///automatically generated by the FlatBuffers compiler, do not modify
///comm\datalayer
{attribute 'conditionalshow' := ''}
METHOD verifyProgressData : BOOL
VAR_INPUT
	data: POINTER TO BYTE;
	size: __UXINT;
	pointer_: UDINT;
END_VAR
VAR
	_bb: ByteBuffer;
	verifier: flatbuffers.Verifier;
	vt_start: UDINT;
	vt_size: UDINT;
END_VAR
_bb(data:=data, _capacity:=TO_UDINT(size));
IF pointer_ = 0 THEN
    verifyProgressData := TRUE;
    RETURN;
END_IF

if pointer_ > (size - SIZEOF(UDINT)) then
    verifyProgressData := FALSE;
    return;
END_IF

vt_start := _bb.getUDINT(pointer_);
if (pointer_ - vt_start) > (size - SIZEOF(UDINT)) then
    verifyProgressData := FALSE;
    return;
END_IF

vt_size := _bb.getUINT(pointer_ - vt_start);
verifier(data:=data, size:=size, pointer_:=pointer_, v_size:=vt_size);

IF verifier.verifyTable() AND verifier.verifyString(4) AND verifier.verifyString(6) THEN
    verifyProgressData := TRUE;
ELSE
    verifyProgressData := FALSE;
END_IF
END_METHOD

END_FUNCTION_BLOCK

// InternHelpers/DCBrowseForFile
{attribute 'hide'}
FUNCTION_BLOCK DCBrowseForFile
VAR_INPUT
	bExecute: BOOL;
	sFileName: STRING;
END_VAR
VAR_OUTPUT
	bDone: BOOL;
	bActive: BOOL;
	bError: BOOL;
	bFound: BOOL;
	ErrorID: CXA_Datalayer.ERROR_CODE;
	ErrorIdent: CXA_Datalayer.ERROR_STRUCT;
END_VAR
VAR
	_dlBrowse: CXA_DATALAYER.DL_BrowseNode;
	_sPath: STRING := S_PARAM_PATH;
	_uiState: UINT;
	_uiNextState: UINT;
	_i: UDINT;
END_VAR
VAR CONSTANT
	S_PARAM_PATH: STRING := 'driveconnect/filesystem/parameterfiles';
	STATE_IDLE: UINT := 0;
	STATE_BROWSE: UINT := 1;
	STATE_CHECK: UINT := 2;
	STATE_DONE: UINT := 3;
	STATE_ERROR: UINT := 4;
END_VAR

CASE _uiState OF 
	STATE_IDLE: 
		IF bExecute THEN 
			_uiNextState := STATE_BROWSE; 
		END_IF
	STATE_BROWSE: 
		IF _dlBrowse.Error THEN 
			ErrorID := _dlBrowse.ErrorID; 
			ErrorIdent := _dlBrowse.ErrorIdent; 
			_uiNextState := STATE_ERROR; 
		ELSIF _dlBrowse.Done THEN 
			_uiNextState := STATE_CHECK; 
		END_IF
	STATE_CHECK: 
		_uiNextState := STATE_DONE; 
	STATE_DONE, STATE_ERROR: 
		IF NOT bExecute THEN 
			_uiNextState := STATE_IDLE; 
		END_IF
END_CASE
_uiState := _uiNextState; 
CASE _uiState OF 
	STATE_IDLE: 
		_dlBrowse.Execute := FALSE; 
		bFound := FALSE; 
	STATE_BROWSE: 
		_dlBrowse.Execute := TRUE;  
	STATE_CHECK:
		_i := 0;
		WHILE _i < _dlBrowse.ChildNum DO 
			IF sFileName = _dlBrowse.GetChildName(_i) THEN 
				bFound := TRUE; 
				EXIT; 
			END_IF
			_i := _i+1; 
		END_WHILE
END_CASE
bDone := _uiState = STATE_DONE; 
bActive := _uiState = STATE_BROWSE OR _uiState = STATE_CHECK; 
bError :=  _uiState = STATE_ERROR; 
_dlBrowse(NodeName := _sPath);

END_FUNCTION_BLOCK

// DriveParamRestore
FUNCTION_BLOCK DriveParamRestore
VAR_INPUT
	bExecute: BOOL;
	sDriveConnectName: STRING;
	iSubDevice: UINT;
	sFileName: STRING;
	iSetIndex: INT;
END_VAR
VAR_OUTPUT
	bDone: BOOL;
	bActive: BOOL;
	bError: BOOL;
	uiProgress: UDINT;
	enTaskState: comm_datalayer_ProgramTaskState;
	ErrorCause: EN_DRIVE_BACKUP_RESTORE_ERROR;
	ErrorID: CXA_Datalayer.ERROR_CODE;
	ErrorIdent: CXA_Datalayer.ERROR_STRUCT;
	sFailureInfo: STRING;
END_VAR
VAR
	_builder: Flatbuffers.FlatBufferBuilder;
	_retoreReq: comm_drive_importParameter_ImportParameter;
	_taskStatus: comm_Datalayer_ProgramTask;
	_pRespString: POINTER TO STRING(255);
	_sRespString: STRING(255);
	_dlCreateNode: CXA_DataLayer.DL_CreateNodeValue;
	_dlReadNode: CXA_DataLayer.DL_ReadNodeValue;
	_dlRestoreReq: CXA_DataLayer.DL_NodeValue;
	_dlTaskPath: CXA_DataLayer.DL_NodeValue;
	_dlTaskResp: CXA_Datalayer.DL_NodeValue;
	_uiState: UINT;
	_uiNextState: UINT;
	_enTaskState: comm_datalayer_ProgramTaskState;
	_sReqString: STRING(255);
	_sBackupFile: STRING(255);
	_uiOffset: UDINT;
	_browseForFile: DCBrowseForFile;
END_VAR
VAR CONSTANT
	STATE_IDLE: UINT := 0;
	STATE_FIND_FILE: UINT := 1;
	STATE_REQ: UINT := 2;
	STATE_RESTORING: UINT := 3;
	STATE_DONE: UINT := 4;
	STATE_ERROR: UINT := 5;
	S_PATH_DEVICES: STRING := 'devices/drives/';
	S_PATH_BACKUPS: STRING := 'filesystem/parameterfiles/';
END_VAR

CASE _uiState OF 
	STATE_IDLE: 
		IF bExecute THEN 
			_uiNextState := STATE_FIND_FILE; 
		END_IF
	STATE_FIND_FILE: 
		IF _browseForFile.bError THEN 
			ErrorID := _browseForFile.ErrorID; 
			ErrorIdent := _browseForFile.ErrorIdent; 
			ErrorCause :=EN_DRIVE_BACKUP_RESTORE_ERROR.FileBrowseFailed; 
			_uiNextState := STATE_ERROR; 
		ELSIF _browseForFile.bDone THEN 
			IF NOT _browseForFile.bFound THEN 
				ErrorCause := EN_DRIVE_BACKUP_RESTORE_ERROR.FileNotFound; 
				_uiNextState := STATE_ERROR; 
			ELSE 
				_uiNextState := STATE_REQ; 
			END_IF;  
		END_IF
	STATE_REQ: 
		IF _dlCreateNode.Error THEN 
			_uiNExtState := STATE_ERROR; 
			ErrorID := _dlCreateNode.ErrorID;
			ErrorIDent := _dlCreateNode.ErrorIdent; 
			ErrorCause := EN_DRIVE_BACKUP_RESTORE_ERROR.RequestFailed;  
		ELSIF _dlCreateNode.Done THEN 
			_uiNextState := STATE_RESTORING; 
		END_IF
	STATE_RESTORING: 
		IF _dlReadNode.Error THEN 
			_uiNextState := STATE_ERROR; 
			ErrorID := _dlReadNode.ErrorID;
			ErrorIDent := _dlReadNode.ErrorIdent; 
			ErrorCause := EN_DRIVE_BACKUP_RESTORE_ERROR.ProgressReadFailed;  
		ELSIF _dlReadNode.Done THEN 
			IF _enTaskState = comm_datalayer_ProgramTaskState.failed THEN 
				_uiNextState := STATE_ERROR; 
				ErrorID := _dlReadNode.ErrorID;
				ErrorIdent := _dlReadNode.ErrorIdent; 
				ErrorCause := EN_DRIVE_BACKUP_RESTORE_ERROR.RestoreFailed;  
				sFailureInfo := _taskStatus.getProgressInfo(); 
			ELSIF _enTaskState = comm_datalayer_ProgramTaskState.done THEN 
				_uiNextState := STATE_DONE; 
			ELSE
				_dlReadNode(Execute := FALSE); 
			END_IF
		END_IF
	STATE_DONE, STATE_ERROR: 
		IF NOT bExecute THEN 
			_uiNextState := STATE_IDLE; 
		END_IF
END_CASE
_uiState := _uiNextState; 
CASE _uiState OF 
	STATE_IDLE: 
		_dlReadNode.Execute := FALSE; 
		_dlCreateNode.Execute := FALSE; 
		_browseForFile.bExecute := FALSE; 
		sFailureInfo := 'OK'; 
		enTaskState := comm_datalayer_ProgramTaskState.done; 
		ErrorCause := EN_DRIVE_BACKUP_RESTORE_ERROR.OK; 
		uiProgress := 0; 
		
	STATE_FIND_FILE: 
		_browseForFile.sFileName := sFileName; 
		_browseForFile.bExecute := TRUE; 
				
	STATE_REQ: 
		_dlCreateNode.Execute := TRUE; 
		_builder(forceDefaults := TRUE); 
		_sBackupFile := CONCAT(S_PATH_BACKUPS,sFileName); 
		_sReqString := CONCAT(S_PATH_DEVICES,sDriveConnectName); 
		_sReqString := CONCAT(_sReqString,'/subdevices/subdevice-'); 
		_sReqString := CONCAT(_sReqString,INT_TO_STRING(iSubDevice)); 
		_sReqString := CONCAT(_sReqString,'/import-parameter'); 
		_uiOffset := _retoreReq.createImportParameter(builder := _builder,fileName := _sBackupFile, setIndex :=iSetIndex);
 		_builder.finish(_uiOffset); 
		_dlRestoreReq.SetFlatbuffer(_builder); 
	STATE_RESTORING: 
		_pRespString := _dlTaskPath.GetData(); 
		_sRespString := _pRespString^; 
		_dlReadNode.Execute := TRUE; 
END_CASE

_dlCreateNode(NodeName := _sReqString,
			  NodeValueIn := _dlRestoreReq, 
			  NodeValueOut := _dlTaskPath); 
			  
_dlReadNode(NodeName := _sRespString,
			NodeValue := _dlTaskResp); 
			
_browseForFile(); 


IF _dlReadNode.Done THEN 
	_taskStatus.getRootAsProgramTask(_dlTaskResp.GetData(),_dlTaskResp.GetSize()); 
	_enTaskState := _taskStatus.getState(); 
	uiProgress := _taskStatus.getProgress(); 
	enTaskState := _enTaskState; 
END_IF

bActive := _uiState <> STATE_IDLE AND _uiState <> STATE_DONE AND _uiState <> STATE_ERROR; 
bDone := _uiState = STATE_DONE; 
bError := _uiState = STATE_ERROR;

END_FUNCTION_BLOCK

// InternHelpers/comm_drive_importParameter_ImportParameter
///automatically generated by the FlatBuffers compiler, do not modify
///comm\drive\importParameter
///Import FlatBuffers Library
FUNCTION_BLOCK comm_drive_importParameter_ImportParameter EXTENDS flatbuffers.Table
VAR
	_builder: REFERENCE TO flatbuffers.FlatBufferBuilder;
	_bb: flatbuffers.ByteBuffer;
END_VAR

///automatically generated by the FlatBuffers compiler, do not modify
///comm\drive\importParameter
///
///Set the values of a ImportParameter and return it.
{attribute 'conditionalshow' := ''}
METHOD _assign : comm_drive_importParameter_ImportParameter
VAR_INPUT
	i: UDINT;
	_bb: REFERENCE TO flatbuffers.ByteBuffer;
END_VAR
_init(i:=i, _bb:=_bb);
_assign:=this^;
END_METHOD

///automatically generated by the FlatBuffers compiler, do not modify
///comm\drive\importParameter
///
///Set the values of a table.
{attribute 'conditionalshow' := ''}
METHOD _init
VAR_INPUT
	i: UDINT;
	_bb: REFERENCE TO flatbuffers.ByteBuffer;
END_VAR
_reset(i:=i, _bb:=_bb);
END_METHOD

///automatically generated by the FlatBuffers compiler, do not modify
///comm\drive\importParameter
///
///Add values to the table.
METHOD addFileName
VAR_INPUT
	fileNameOffset: UDINT;
END_VAR
IF NOT __ISVALIDREF(_builder) THEN
  SysExceptGenerateException(RTSEXCPT_INVALID_HANDLE);
END_IF
_builder.add_Offset(o:=0, x:=fileNameOffset, d:=0);
END_METHOD

///automatically generated by the FlatBuffers compiler, do not modify
///comm\drive\importParameter
///
///Add values to the table.
METHOD addSetIndex
VAR_INPUT
	setIndex: DINT;
END_VAR
IF NOT __ISVALIDREF(_builder) THEN
  SysExceptGenerateException(RTSEXCPT_INVALID_HANDLE);
END_IF
_builder.add_DINT(o:=1, x:=setIndex, d:=0);
END_METHOD

///automatically generated by the FlatBuffers compiler, do not modify
///comm\drive\importParameter
///
///Creates a table in the Flatbuffer and returns the offset to it.
METHOD createImportParameter : UDINT
VAR_INPUT
	builder: REFERENCE TO flatbuffers.FlatBufferBuilder;
	fileName: STRING;
	setIndex: DINT;
END_VAR
VAR
	fileNameOffset: UDINT;
END_VAR
_builder REF= builder;
IF NOT __ISVALIDREF(_builder) THEN
  SysExceptGenerateException(RTSEXCPT_INVALID_HANDLE);
END_IF
fileNameOffset := builder.createString(fileName);
_builder.startTable(numfields:=2);
addFileName(fileNameOffset:=fileNameOffset);
addSetIndex(setIndex:=setIndex);
createImportParameter := endImportParameter();
END_METHOD

///automatically generated by the FlatBuffers compiler, do not modify
///comm\drive\importParameter
///
///End the table and return a offset to it
METHOD endImportParameter : UDINT
VAR
	o: UDINT;
END_VAR
o := _builder.endTable();
_builder REF= 0;
endImportParameter := o;
END_METHOD

///automatically generated by the FlatBuffers compiler, do not modify
///comm\drive\importParameter
///
///Returns a String.
METHOD getFileName : STRING
VAR
	o: UDINT;
END_VAR
o := _offset(vtable_offset:=4);
IF o<>0 THEN
    getFileName := _string(offset:=o+bb_pos);
ELSE
    getFileName := '';
END_IF
END_METHOD

///automatically generated by the FlatBuffers compiler, do not modify
///comm\drive\importParameter
///
///Returns a String as pointer to byte.
METHOD getFileNameAsBytePtr : POINTER TO BYTE
VAR
	o: UDINT;
END_VAR
o := _offset(vtable_offset:=4);
IF o<>0 THEN
    getFileNameAsBytePtr := _stringPtr(offset:=o+bb_pos);
ELSE
    getFileNameAsBytePtr := 0;
END_IF
END_METHOD

///automatically generated by the FlatBuffers compiler, do not modify
///comm\drive\importParameter
///
///Returns a ImportParameter from the ByteBuffer.
/// 
METHOD getRootAsImportParameter : comm_drive_importParameter_ImportParameter
VAR_INPUT
	data: POINTER TO BYTE;
	size: __UXINT;
END_VAR
_bb(data:=data, _capacity:=TO_UDINT(size));
bb REF= _bb;
getRootAsImportParameter := _assign(i:=bb.getUDINT(0), _bb:=bb);
END_METHOD

///automatically generated by the FlatBuffers compiler, do not modify
///comm\drive\importParameter
///
///Returns a DINT from the table.
METHOD getSetIndex : DINT
VAR
	o: UDINT;
END_VAR
o := _offset(vtable_offset:=6);
IF o<>0 THEN
    getSetIndex := bb.getDINT(offset:=o+bb_pos);
ELSE
    getSetIndex := 0;
END_IF
END_METHOD

///automatically generated by the FlatBuffers compiler, do not modify
///comm\drive\importParameter
///
///Start the table to add values.
METHOD startImportParameter
VAR_INPUT
	builder: REFERENCE TO flatbuffers.FlatBufferBuilder;
END_VAR
_builder REF= builder;
_builder.startTable(numfields:=2);
END_METHOD

///automatically generated by the FlatBuffers compiler, do not modify
///comm\drive\importParameter
METHOD verify : BOOL
VAR_INPUT
	data: POINTER TO BYTE;
	size: __UXINT;
END_VAR
VAR
	_bb: ByteBuffer;
END_VAR
_bb(data:=data, _capacity:=TO_UDINT(size));
verify := verifyImportParameter(data, size, _bb.getUDINT(0));
END_METHOD

///automatically generated by the FlatBuffers compiler, do not modify
///comm\drive\importParameter
{attribute 'conditionalshow' := ''}
METHOD verifyImportParameter : BOOL
VAR_INPUT
	data: POINTER TO BYTE;
	size: __UXINT;
	pointer_: UDINT;
END_VAR
VAR
	_bb: ByteBuffer;
	verifier: flatbuffers.Verifier;
	vt_start: UDINT;
	vt_size: UDINT;
END_VAR
_bb(data:=data, _capacity:=TO_UDINT(size));
IF pointer_ = 0 THEN
    verifyImportParameter := TRUE;
    RETURN;
END_IF

if pointer_ > (size - SIZEOF(UDINT)) then
    verifyImportParameter := FALSE;
    return;
END_IF

vt_start := _bb.getUDINT(pointer_);
if (pointer_ - vt_start) > (size - SIZEOF(UDINT)) then
    verifyImportParameter := FALSE;
    return;
END_IF

vt_size := _bb.getUINT(pointer_ - vt_start);
verifier(data:=data, size:=size, pointer_:=pointer_, v_size:=vt_size);

IF verifier.verifyTable() AND verifier.verifyString(4) AND verifier.verifyScalar(6) THEN
    verifyImportParameter := TRUE;
ELSE
    verifyImportParameter := FALSE;
END_IF
END_METHOD

END_FUNCTION_BLOCK

// License_And_Use
(*
Copyright  2025 Riley Duffy

Permission is hereby granted, free of charge, to any person obtaining a copy of this software and associated documentation files
the “Software”), to deal in the Software without restriction, including without limitation the rights to use, copy, modify, merge,
publish, distribute, sublicense, and/or sell copies of the Software, and to permit persons to whom the Software is furnished to do so,
subject to the following conditions:

The above copyright notice and this permission notice shall be included in all copies or substantial portions of the Software.

THE SOFTWARE IS PROVIDED “AS IS”, WITHOUT WARRANTY OF ANY KIND, EXPRESS OR IMPLIED,
 INCLUDING BUT NOT LIMITED TO THE WARRANTIES OF MERCHANTABILITY, FITNESS FOR A PARTICULAR PURPOSE AND NONINFRINGEMENT.
 IN NO EVENT SHALL THE AUTHORS OR COPYRIGHT HOLDERS BE LIABLE FOR ANY CLAIM, DAMAGES OR OTHER LIABILITY,
 WHETHER IN AN ACTION OF CONTRACT, TORT OR OTHERWISE, ARISING FROM, OUT OF OR IN CONNECTION WITH THE SOFTWARE
 OR THE USE OR OTHER DEALINGS IN THE SOFTWARE.*)
FUNCTION_BLOCK License_And_Use
VAR_INPUT
END_VAR
VAR_OUTPUT
END_VAR
VAR
END_VAR

(*
Copyright  2025 Riley Duffy

Permission is hereby granted, free of charge, to any person obtaining a copy of this software and associated documentation files
(the “Software”), to deal in the Software without restriction, including without limitation the rights to use, copy, modify, merge,
publish, distribute, sublicense, and/or sell copies of the Software, and to permit persons to whom the Software is furnished to do so,
subject to the following conditions:

The above copyright notice and this permission notice shall be included in all copies or substantial portions of the Software.

THE SOFTWARE IS PROVIDED “AS IS”, WITHOUT WARRANTY OF ANY KIND, EXPRESS OR IMPLIED,
 INCLUDING BUT NOT LIMITED TO THE WARRANTIES OF MERCHANTABILITY, FITNESS FOR A PARTICULAR PURPOSE AND NONINFRINGEMENT.
 IN NO EVENT SHALL THE AUTHORS OR COPYRIGHT HOLDERS BE LIABLE FOR ANY CLAIM, DAMAGES OR OTHER LIABILITY,
 WHETHER IN AN ACTION OF CONTRACT, TORT OR OTHERWISE, ARISING FROM, OUT OF OR IN CONNECTION WITH THE SOFTWARE
 OR THE USE OR OTHER DEALINGS IN THE SOFTWARE.*)

END_FUNCTION_BLOCK
